// SIMATIC S7-200 project (STEP 7-Micro/WIN), CPU 226 REL 01.23

ORGANIZATION_BLOCK MAIN:OB1
TITLE=[Project Introduction]
// This code is a control system designed for the finished product delivery line of Lenovo brand, which is used for production line control.
// The system is booted with I0.0 (requires M0.0 to take effect with I0.3 or already set).
// [Hardware]
// The equipment involved in the system includes conveyor belts and diverters.
// [Code Comments]
// The entire process begins with the activation of Start Button 1. The System Ready Flag is set when either the Reset Button is pressed or the Emergency Stop Button is not engaged, indicating the system enters standby mode.
// 
// After conveyor startup, Inlet Valve A1 opens under the following conditions:
// 
// The Feed Enable Flag or Feed Delay Timer is active,
// 
// Start Button 1 is released,
// 
// AND either Midpoint Sensor 1 or Divert Path Sensor 1 detects products.
// 
// The Feed Enable Flag is set when either Inlet Valve A Feedback 2 or Inlet Valve B Feedback 2 confirms valve opening, AND Cooler Feedback 1 does not detect full liquid level to prevent overflow.
// 
// Inlet Valve B1 activates when:
// 
// Midpoint Sensor 2 detects products,
// 
// Low Level Flag is inactive,
// 
// AND either Midpoint Sensor 1 or Divert Path Sensor 1 detects products (prevents incorrect diverter operation).
// 
// The Low Level Flag is set when Level Sensor 2 does not detect full capacity AND Inlet Valve B1 remains closed.
// 
// During transport, Temperature Sensor 2 monitors ambient conditions:
// 
// If temperature is low, Heater 2 activates when:
// 
// Heater Control Flag and Running Indicator 1 are active,
// 
// AND Level Sensor 4 is not at full capacity.
// 
// If temperature is high, Outlet Valve 2 opens when:
// 
// High Temp Flag 2 or Low Temp Flag is active,
// 
// AND Cooler Feedback 3 shows no fault,
// 
// WITH parallel activation of Cooler 2.
// 
// High Temp Flag 2 sets when Level Sensor 3 detects overheating AND Low Temp Flag 2 is inactive. Conversely, Low Temp Flag 2 sets when Level Sensor 3 detects under-temperature AND High Temp Flag 2 is inactive.
// 
// At final processing stage:
// 
// Agitator Motor 2 starts when:
// 
// Agitation Delay Timer or Discharge Enable Flag is active,
// 
// AND Low Level Flag is set.
// 
// Agitation Enable Flag sets when:
// 
// Start Button 1 is pressed,
// 
// Temperature Sensor 2 reads within range,
// 
// AND Inlet Valve B1 is closed.
// 
// Post-agitation, Outlet Valve 1 opens when:
// 
// Stop Button 1 is pressed,
// 
// Manual/Auto Switch 1 is off,
// 
// Start Button 1 is released,
// 
// AND Divert Path Sensor 1 confirms product presence.
// 
// System status is indicated by Running Indicator 2, which illuminates when:
// 
// Cooler 1 operates,
// 
// Start Button 2 is pressed,
// 
// AND System Ready Flag is active.
// 
// Stop Button 1 allows immediate interruption, 
BEGIN
Network 1 // Network Title
// Network Comment
LD     Q1.1
ON     I5.0
A      M0.0
=      Q3.3
Network 2
LD     I0.3
O      M0.0
A      I0.4
=      M0.0
Network 3
LDN    I1.5
LD     I1.5
AN     M7.2
A      M7.0
A      Q1.4
OLD
A      M0.0
=      Q1.5
Network 4
LDN    I1.4
LD     I1.4
LDN    M6.2
A      M6.0
LDN    I4.2
AN     I4.4
OLD
ALD
A      Q1.3
OLD
AN     M9.2
A      M0.0
AN     M9.1
=      Q1.4
Network 5
LDN    I1.3
LD     I1.3
A      Q1.2
OLD
A      M0.0
=      Q1.3
Network 6
LDN    I1.2
LD     I1.2
A      Q3.3
OLD
A      M0.0
=      Q1.2
Network 7
LDN    I1.1
LD     I1.1
A      M5.0
A      Q0.7
OLD
A      I0.0
A      M0.0
=      Q1.1
Network 8
LD     I2.6
A      I2.7
EU
A      I1.1
O      M5.0
A      I0.0
AN     M5.1
A      M0.0
=      M5.0
Network 9
LD     I1.1
ED
=      M5.1
Network 10
LD     I0.7
O      M15.1
A      M0.0
AN     I0.3
=      M15.1
Network 11
LDN    I0.0
A      I0.1
AN     I0.2
LDN    M10.4
A      I0.0
AN     M2.0
AN     M2.1
AN     M2.2
AN     M2.3
OLD
A      M0.0
AN     M10.2
AN     I0.5
AN     M15.1
A      I0.6
=      Q0.7
Network 12
LDN    I0.0
AN     I0.1
A      I0.2
AN     I0.5
A      I0.6
A      M0.0
=      Q1.0
Network 13
LD     I2.5
O      I2.4
A      I1.6
O      M2.0
A      I0.0
A      M0.0
=      M2.0
Network 14
LD     I2.3
A      I2.4
O      M2.1
A      I0.0
A      M0.0
=      M2.1
Network 15
LD     I0.0
A      I1.7
AN     Q0.5
A      M0.0
=      M2.2
Network 16
LDN    I2.1
LD     I2.1
AN     M12.0
A      Q3.5
OLD
A      M0.0
=      Q0.5
Network 17
LDN    I3.3
LD     I3.3
A      Q0.6
OLD
AN     I3.0
LDN    I3.3
LD     I3.3
A      I3.2
AN     M3.0
OLD
LD     I3.3
AN     I3.2
AN     M3.1
A      Q0.6
OLD
A      I3.0
OLD
A      M0.0
AN     I4.6
=      Q3.5
Network 18
LD     I3.3
EU
O      M3.0
A      M12.0
AN     I4.0
A      I3.0
A      M0.0
=      M3.0
Network 19
LD     I3.2
ED
O      M3.1
AN     I4.0
A      M12.0
A      I3.0
A      M0.0
=      M3.1
Network 20
LD     M3.0
O      M3.1
A      M12.0
A      M0.0
=      Q2.4
Network 21
LDN    I2.2
LD     I2.2
A      Q2.3
OLD
A      M0.0
=      Q0.6
Network 22
LDN    I3.4
LDN    M13.0
A      I3.4
A      Q2.2
OLD
A      M0.0
=      Q2.3
Network 23
LDN    I3.6
O      I3.6
AN     I3.1
LDN    I3.6
LD     I3.6
A      I3.5
LDN    M4.0
ON     M13.0
ALD
OLD
LD     I3.6
AN     I3.5
LDN    M4.1
ON     M13.0
ALD
A      Q3.4
OLD
A      I3.1
OLD
AN     I4.7
A      M0.0
=      Q2.2
Network 24
LD     I3.6
EU
O      M4.0
AN     I4.1
A      I3.1
A      M13.0
A      M0.0
=      M4.0
Network 25
LD     I3.5
ED
O      M4.1
AN     I4.1
A      M13.0
A      I3.1
A      M0.0
=      M4.1
Network 26
LD     M4.0
O      M4.1
A      M13.0
A      M0.0
=      Q2.5
Network 27
LDN    I3.7
A      M0.0
=      Q3.4
Network 28
LD     M2.0
O      M2.1
ON     I0.0
ON     I0.6
O      I0.5
=      Q0.4
Network 29
LD     I1.4
O      M6.0
AN     M9.2
AN     M9.1
AN     M6.1
AN     M6.7
A      M0.0
=      M6.0
Network 30
LD     I4.4
ED
A      I1.4
S      M9.1, 1
Network 31
LD     I4.2
EU
R      M9.1, 1
Network 32
LD     I4.4
O      M6.1
AN     M6.0
A      M0.0
AN     M6.7
O      M9.2
=      M6.1
A      Q1.3
=      M7.0
Network 33
LD     M7.0
LD     Q1.3
AN     I4.4
OLD
AN     M9.0
=      Q3.0
Network 34
LD     I1.4
ED
A      I4.4
S      M9.0, 1
Network 35
LD     I4.2
EU
R      M9.0, 1
Network 36
LD     I1.4
ED
O      M6.2
AN     M6.7
=      M6.2
Network 37
LD     T37
EU
A      Q1.3
S      M9.2, 1
Network 38
LD     I1.4
AN     I4.2
A      I4.4
AN     M6.7
A      Q1.3
TON    T37, +30
Network 39
LD     I4.4
ED
R      M9.2, 1
Network 40
LD     I4.2
EU
=      M6.7
Network 41
LD     I1.5
AN     I4.3
O      M7.0
AN     M7.1
AN     M7.3
A      M0.0
=      M7.0
Network 42
LD     I4.5
AN     I4.3
O      M7.1
AN     M7.0
A      M0.0
AN     M7.3
=      M7.1
A      Q1.4
=      Q3.1
Network 43
LD     I1.5
ED
O      M7.2
AN     M7.3
=      M7.2
Network 44
LD     I4.3
ED
=      M7.3
Network 45
LD     I1.7
O      M10.0
AN     M10.1
A      M0.0
=      M10.0
Network 46
LD     M10.0
A      I2.3
=      M10.1
Network 47
LD     I2.0
AN     Q0.5
=      M10.2
Network 48
LD     I1.7
A      I2.0
A      M0.0
=      M10.4
Network 49
LD     I2.1
O      M11.0
AN     M11.4
A      M0.0
A      I5.4
=      M11.0
Network 50
LD     M11.0
A      I1.0
O      M11.1
AN     M11.4
A      I5.4
A      M0.0
=      M11.1
Network 51
LD     M11.0
A      I3.2
A      I2.1
O      M11.2
A      M0.0
A      I5.4
AN     M11.4
=      M11.2
Network 52
LD     I3.2
ED
=      M11.3
Network 53
LD     I3.3
ED
=      M11.4
Network 54
LD     M11.2
O      M11.1
A      I5.4
A      M0.0
=      M12.0
Network 55
LD     I3.4
O      M13.1
A      M0.0
AN     M13.2
AN     M12.5
=      M13.1
Network 56
LD     M13.1
AN     I3.4
AN     I3.5
O      M12.1
AN     M12.5
=      M12.1
Network 57
LD     I3.5
A      I3.6
A      M4.1
O      M12.2
AN     M12.3
=      M12.2
Network 58
LD     I3.4
ED
=      M13.2
Network 59
LD     M13.1
A      I5.6
O      M12.4
AN     M12.5
=      M12.4
Network 60
LD     I3.6
ED
=      M12.5
Network 61
LD     M12.1
AN     M12.4
=      M13.0
END_ORGANIZATION_BLOCK
